Staubli VAL3: Safety.pgx

program Safety()
begin

  //同步任务来实现安全检测
  while true
    //获取速度
    nRobotSpeed=getSpeed(tTool)


    //判断位置是否超过安全区域
    pCurrent=here(tTool,world)
    if distance(pCurrent.trsf,trSafety)>200
      if isPowered()
        popUpMsg("超过安全限制")
        disablePower()
      endIf
    endIf
    delay(0)
  endWhile


end
